(* Logix 5000 project; controller STAT 1756-L72 rev 20.12; software revision 20.04; part 17 of 34 *)
(* tags used below, declared in another part *)
   B14 : DINT[30];
   B16 : DINT[30];
   B17 : DINT[30];
   B3 : DINT[256];
   B9 : DINT[40];
   I7_000_Bit08 : ALIAS FOR I7[0].8;   // midden alarm ketel tampon
   I8_000_Bit09 : ALIAS FOR I8[0].9;   // midden niveau kuip 1 voorb. polyelectrolute
   I8_000_Bit10 : ALIAS FOR I8[0].10;   // hoog niveau kuip 1 voorb. polyelectrolute
   I8_000_Bit12 : ALIAS FOR I8[0].12;   // midden niveau kuip 2 voorb. polyelectrolute
   I8_000_Bit13 : ALIAS FOR I8[0].13;   // hoog niveau pekel
   N26 : DINT[256];
   O12_001_Bit06 : ALIAS FOR O12[1].6;   // TFB1_1_EV1 TFB1_1_EV1
   O12_001_Bit07 : ALIAS FOR O12[1].7;   // TFB1_1_EV2 TFB1_1_EV2
   O12_001_Bit08 : ALIAS FOR O12[1].8;   // TFB1_2_EV3 TFB1_2_EV3
   O12_001_Bit09 : ALIAS FOR O12[1].9;   // TFB1_2_EV4 TFB1_2_EV4
   O12_001_Bit10 : ALIAS FOR O12[1].10;   // TFB1_2_EV10 TFB1_2_EV10
   O12_001_Bit11 : ALIAS FOR O12[1].11;   // TFB1_EV9 TFB1_EV9
   O12_001_Bit12 : ALIAS FOR O12[1].12;   // TFB1_2_EV5 TFB1_2_EV5
   O12_001_Bit13 : ALIAS FOR O12[1].13;   // TFB1_2_EV6 TFB1_2_EV6
   O13_001_Bit10 : ALIAS FOR O13[1].10;   // TFB1_2_EV7 TFB1_2_EV7
   O13_001_Bit11 : ALIAS FOR O13[1].11;   // TFB1_2_EV8 TFB1_2_EV8
   O13_001_Bit12 : ALIAS FOR O13[1].12;   // TFB1_2_EV11 TFB1_2_EV11
   O15_000_Bit09 : ALIAS FOR O15[0].9;   // CLEAN_V11 CLEAN_V11
   O15_000_Bit10 : ALIAS FOR O15[0].10;   // CLEAN_V12 CLEAN_V12
   O15_000_Bit11 : ALIAS FOR O15[0].11;   // CLEAN_V13 CLEAN_V13
   O15_000_Bit12 : ALIAS FOR O15[0].12;   // CLEAN_V14 CLEAN_V14
   O15_000_Bit13 : ALIAS FOR O15[0].13;   // CLEAN_V21 CLEAN_V21
   O15_000_Bit14 : ALIAS FOR O15[0].14;   // CLEAN_V22 CLEAN_V22
   O15_000_Bit15 : ALIAS FOR O15[0].15;   // CLEAN_V23 CLEAN_V23
   O15_001_Bit00 : ALIAS FOR O15[1].0;   // CLEAN_V24 CLEAN_V24
   O15_001_Bit01 : ALIAS FOR O15[1].1;   // CLEAN_V3 CLEAN_V3
   O1_011_Bit00 : ALIAS FOR O1[11].0;
   O1_011_Bit03 : ALIAS FOR O1[11].3;
   STEP_REI_Z_2_3_6_7 : BOOL;
   STEP_REI_Z_2_3_6_7B : BOOL;
   STEP_REO_Z_2_6_A_ET_B : BOOL;
   T4 : TIMER[200];
(* ibt, continued *)

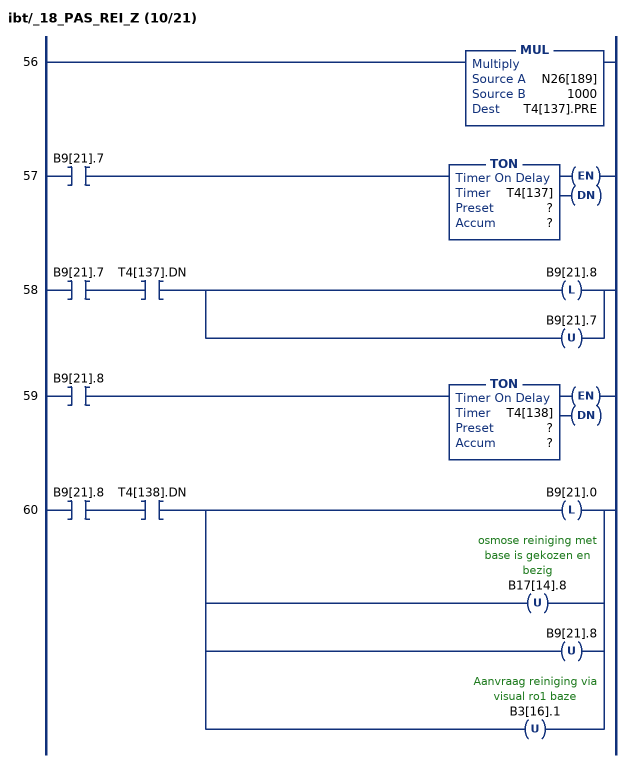
   [picture p297: ibt/_18_PAS_REI_Z rungs 56-60]
   56: MUL(N26[189],1000,T4[137].PRE);
   57: XIC(B9[21].7)TON(T4[137],?,?);
   58: XIC(B9[21].7)XIC(T4[137].DN)[OTL(B9[21].8) ,OTU(B9[21].7) ];
   59: XIC(B9[21].8)TON(T4[138],?,?);
   60: XIC(B9[21].8)XIC(T4[138].DN)[[OTL(B9[21].0) ,OTU(B17[14].8) ] ,[OTU(B9[21].8) ,OTU(B3[16].1) ] ];
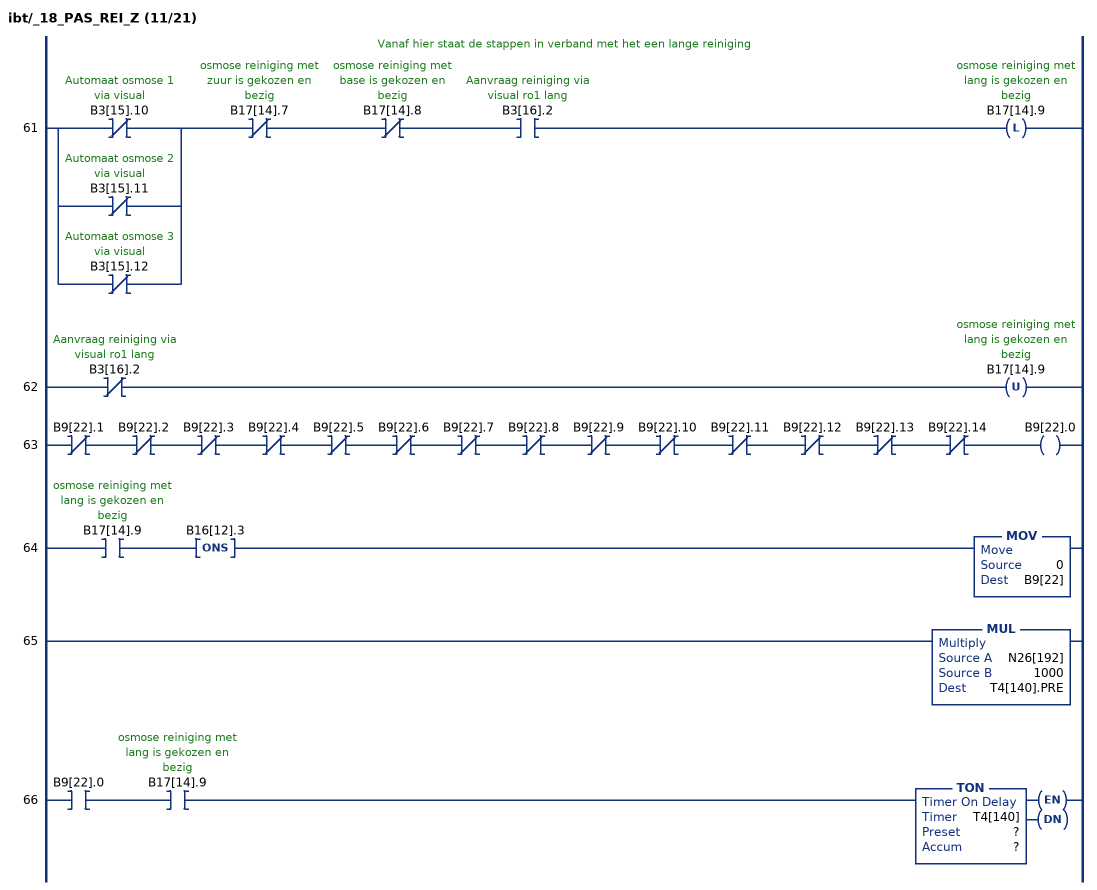
   // Vanaf hier staat de stappen in verband met het een lange reiniging
   61: [XIO(B3[15].10) ,[XIO(B3[15].11) ,XIO(B3[15].12) ] ]XIO(B17[14].7)XIO(B17[14].8)XIC(B3[16].2)OTL(B17[14].9);
   62: XIO(B3[16].2)OTU(B17[14].9);
   63: XIO(B9[22].1)XIO(B9[22].2)XIO(B9[22].3)XIO(B9[22].4)XIO(B9[22].5)XIO(B9[22].6)XIO(B9[22].7)XIO(B9[22].8)XIO(B9[22].9)XIO(B9[22].10)XIO(B9[22].11)XIO(B9[22].12)XIO(B9[22].13)XIO(B9[22].14)OTE(B9[22].0);
   64: XIC(B17[14].9)ONS(B16[12].3)MOV(0,B9[22]);
   65: MUL(N26[192],1000,T4[140].PRE);
   66: XIC(B9[22].0)XIC(B17[14].9)TON(T4[140],?,?);
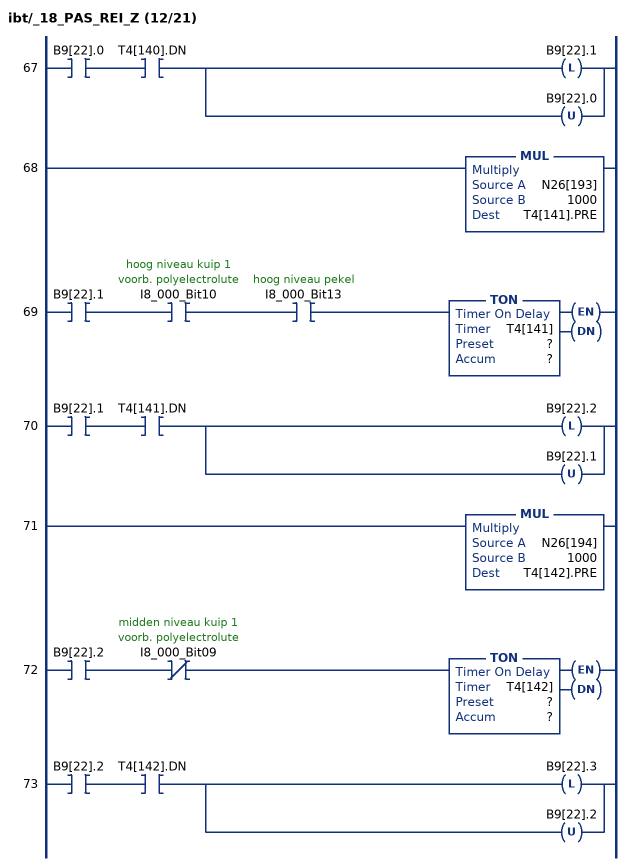
   67: XIC(B9[22].0)XIC(T4[140].DN)[OTL(B9[22].1) ,OTU(B9[22].0) ];
   68: MUL(N26[193],1000,T4[141].PRE);
   69: XIC(B9[22].1)XIC(I8_000_Bit10)XIC(I8_000_Bit13)TON(T4[141],?,?);
   70: XIC(B9[22].1)XIC(T4[141].DN)[OTL(B9[22].2) ,OTU(B9[22].1) ];
   71: MUL(N26[194],1000,T4[142].PRE);
   72: XIC(B9[22].2)XIO(I8_000_Bit09)TON(T4[142],?,?);
   73: XIC(B9[22].2)XIC(T4[142].DN)[OTL(B9[22].3) ,OTU(B9[22].2) ];
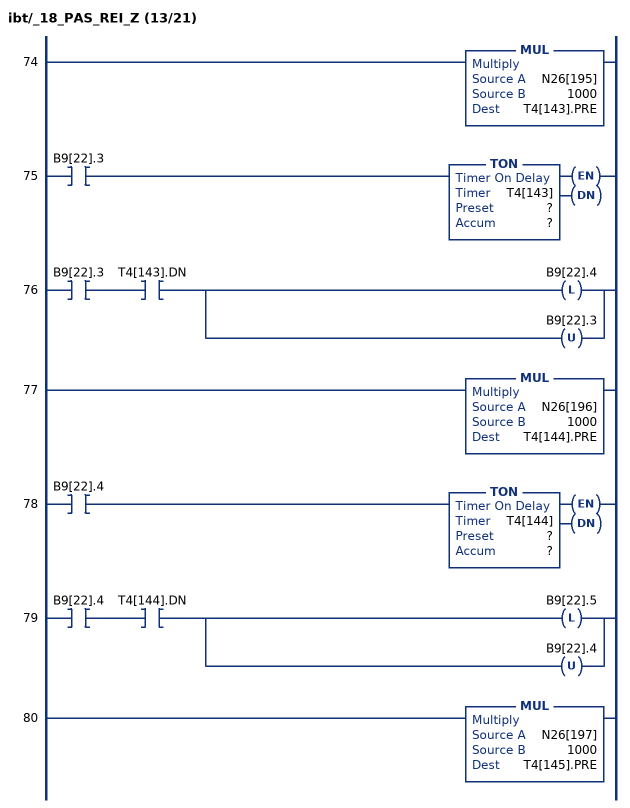
   74: MUL(N26[195],1000,T4[143].PRE);
   75: XIC(B9[22].3)TON(T4[143],?,?);
   76: XIC(B9[22].3)XIC(T4[143].DN)[OTL(B9[22].4) ,OTU(B9[22].3) ];
   77: MUL(N26[196],1000,T4[144].PRE);
   78: XIC(B9[22].4)TON(T4[144],?,?);
   79: XIC(B9[22].4)XIC(T4[144].DN)[OTL(B9[22].5) ,OTU(B9[22].4) ];
   80: MUL(N26[197],1000,T4[145].PRE);
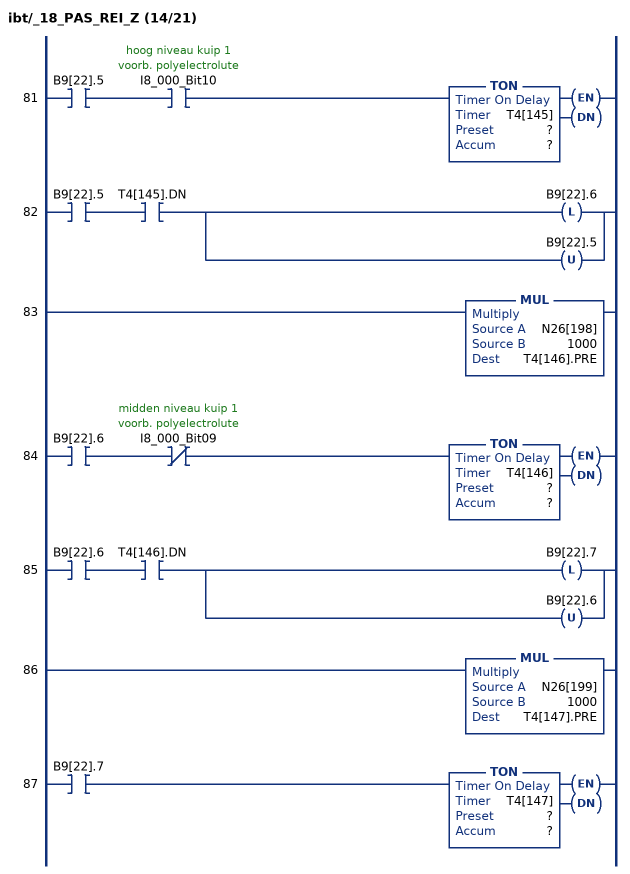
   81: XIC(B9[22].5)XIC(I8_000_Bit10)TON(T4[145],?,?);
   82: XIC(B9[22].5)XIC(T4[145].DN)[OTL(B9[22].6) ,OTU(B9[22].5) ];
   83: MUL(N26[198],1000,T4[146].PRE);
   84: XIC(B9[22].6)XIO(I8_000_Bit09)TON(T4[146],?,?);
   85: XIC(B9[22].6)XIC(T4[146].DN)[OTL(B9[22].7) ,OTU(B9[22].6) ];
   86: MUL(N26[199],1000,T4[147].PRE);
   87: XIC(B9[22].7)TON(T4[147],?,?);
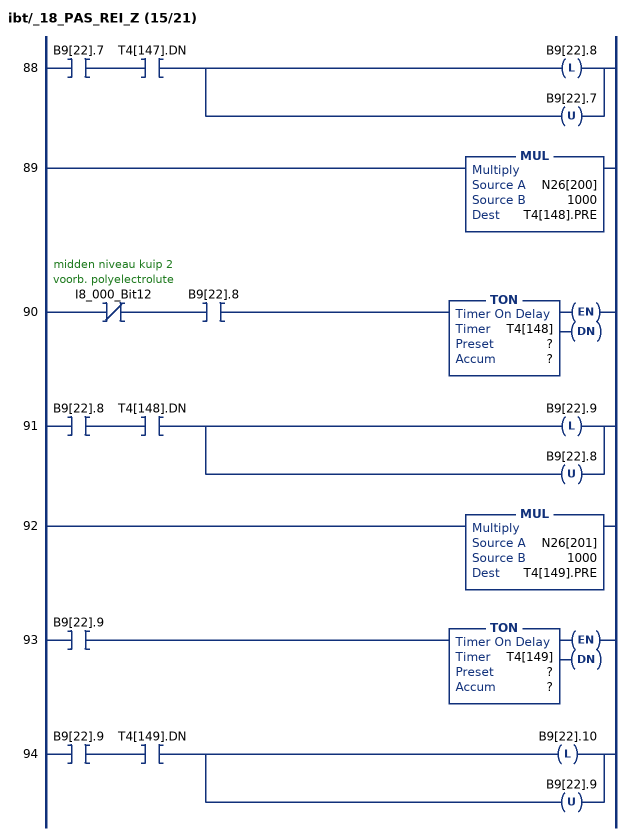
   88: XIC(B9[22].7)XIC(T4[147].DN)[OTL(B9[22].8) ,OTU(B9[22].7) ];
   89: MUL(N26[200],1000,T4[148].PRE);
   90: XIO(I8_000_Bit12)XIC(B9[22].8)TON(T4[148],?,?);
   91: XIC(B9[22].8)XIC(T4[148].DN)[OTL(B9[22].9) ,OTU(B9[22].8) ];
   92: MUL(N26[201],1000,T4[149].PRE);
   93: XIC(B9[22].9)TON(T4[149],?,?);
   94: XIC(B9[22].9)XIC(T4[149].DN)[OTL(B9[22].10) ,OTU(B9[22].9) ];
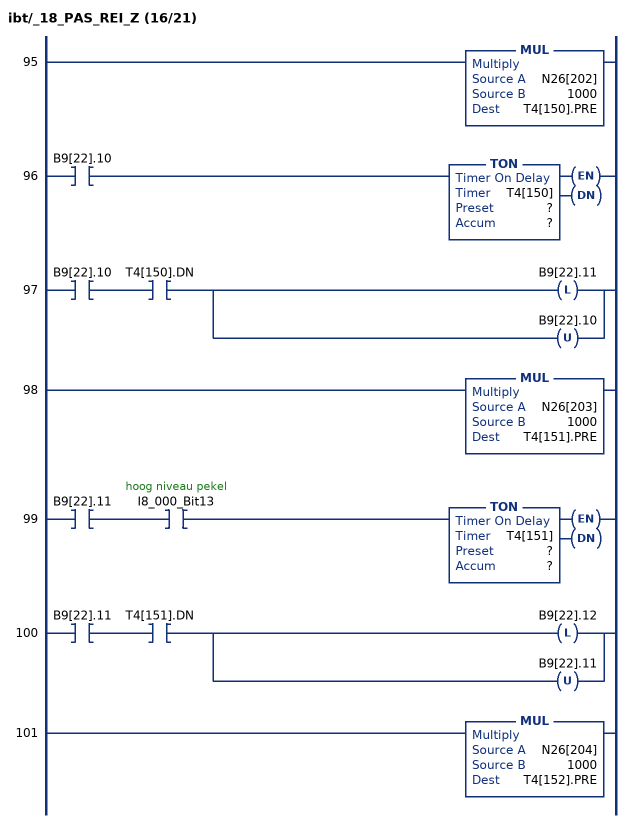
   95: MUL(N26[202],1000,T4[150].PRE);
   96: XIC(B9[22].10)TON(T4[150],?,?);
   97: XIC(B9[22].10)XIC(T4[150].DN)[OTL(B9[22].11) ,OTU(B9[22].10) ];
   98: MUL(N26[203],1000,T4[151].PRE);
   99: XIC(B9[22].11)XIC(I8_000_Bit13)TON(T4[151],?,?);
   100: XIC(B9[22].11)XIC(T4[151].DN)[OTL(B9[22].12) ,OTU(B9[22].11) ];
   101: MUL(N26[204],1000,T4[152].PRE);
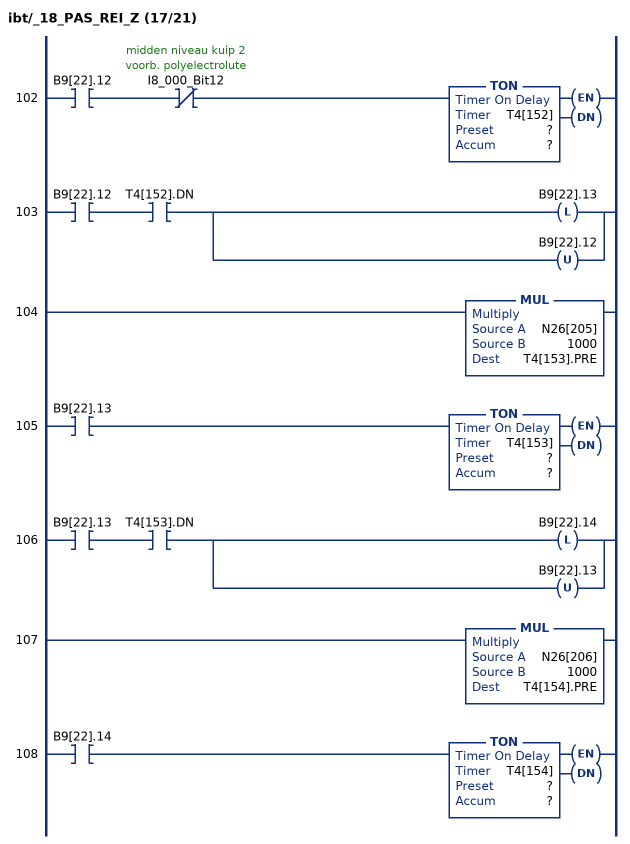
   102: XIC(B9[22].12)XIO(I8_000_Bit12)TON(T4[152],?,?);
   103: XIC(B9[22].12)XIC(T4[152].DN)[OTL(B9[22].13) ,OTU(B9[22].12) ];
   104: MUL(N26[205],1000,T4[153].PRE);
   105: XIC(B9[22].13)TON(T4[153],?,?);
   106: XIC(B9[22].13)XIC(T4[153].DN)[OTL(B9[22].14) ,OTU(B9[22].13) ];
   107: MUL(N26[206],1000,T4[154].PRE);
   108: XIC(B9[22].14)TON(T4[154],?,?);
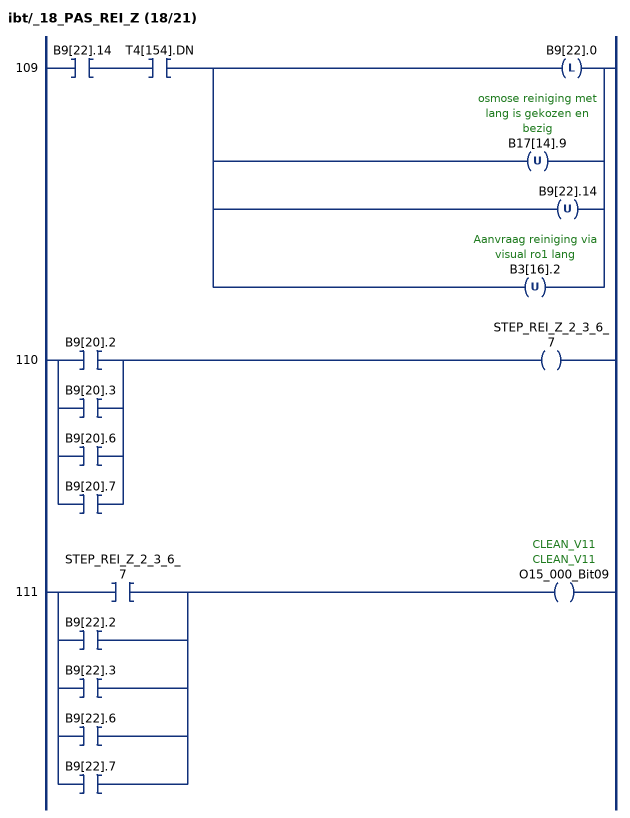
   109: XIC(B9[22].14)XIC(T4[154].DN)[[OTL(B9[22].0) ,OTU(B17[14].9) ] ,[OTU(B9[22].14) ,OTU(B3[16].2) ] ];
   110: [XIC(B9[20].2) ,[XIC(B9[20].3) ,[XIC(B9[20].6) ,XIC(B9[20].7) ] ] ]OTE(STEP_REI_Z_2_3_6_7);
   111: [XIC(STEP_REI_Z_2_3_6_7) ,[[XIC(B9[22].2) ,XIC(B9[22].3) ] ,[XIC(B9[22].6) ,XIC(B9[22].7) ] ] ]OTE(O15_000_Bit09);
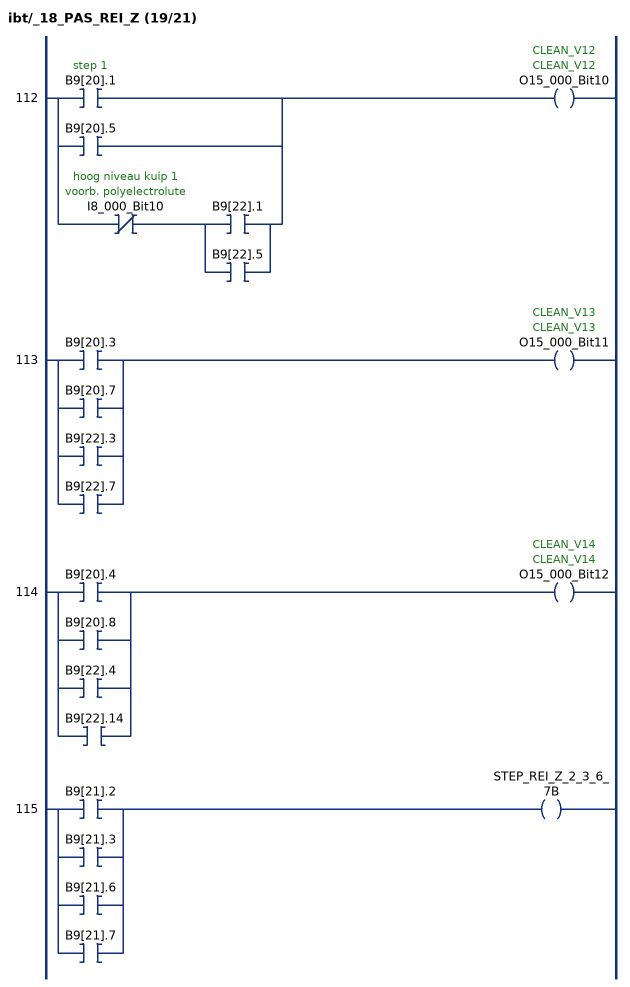
   112: [[XIC(B9[20].1) ,XIC(B9[20].5) ] ,XIO(I8_000_Bit10) [XIC(B9[22].1) ,XIC(B9[22].5) ] ]OTE(O15_000_Bit10);
   113: [[XIC(B9[20].3) ,XIC(B9[20].7) ] ,[XIC(B9[22].3) ,XIC(B9[22].7) ] ]OTE(O15_000_Bit11);
   114: [[XIC(B9[20].4) ,XIC(B9[20].8) ] ,[XIC(B9[22].4) ,XIC(B9[22].14) ] ]OTE(O15_000_Bit12);
   115: [[XIC(B9[21].2) ,XIC(B9[21].3) ] ,[XIC(B9[21].6) ,XIC(B9[21].7) ] ]OTE(STEP_REI_Z_2_3_6_7B);
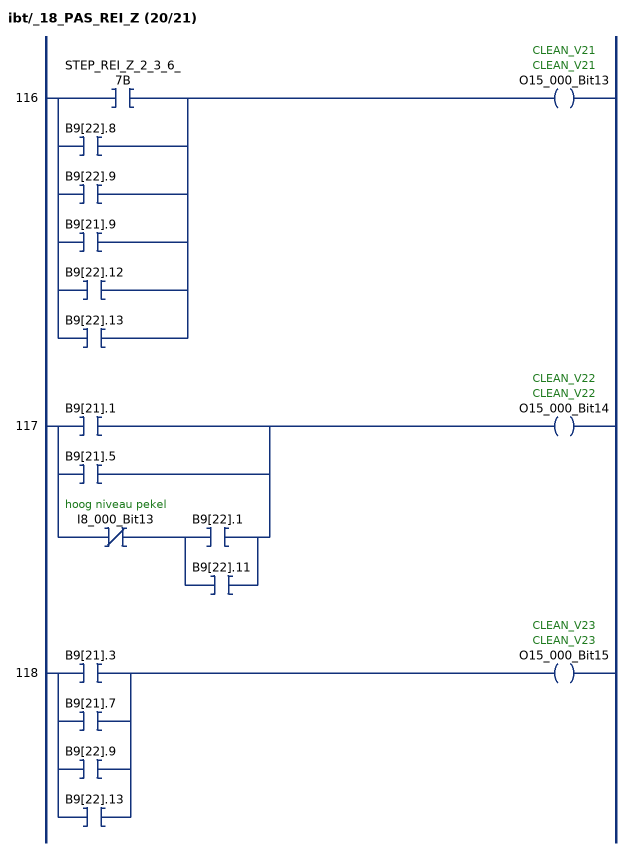
   116: [[XIC(STEP_REI_Z_2_3_6_7B) ,XIC(B9[22].8) ,XIC(B9[22].9) ] ,[XIC(B9[21].9) ,[XIC(B9[22].12) ,XIC(B9[22].13) ] ] ]OTE(O15_000_Bit13);
   117: [[XIC(B9[21].1) ,XIC(B9[21].5) ] ,XIO(I8_000_Bit13) [XIC(B9[22].1) ,XIC(B9[22].11) ] ]OTE(O15_000_Bit14);
   118: [[XIC(B9[21].3) ,XIC(B9[21].7) ] ,[XIC(B9[22].9) ,XIC(B9[22].13) ] ]OTE(O15_000_Bit15);
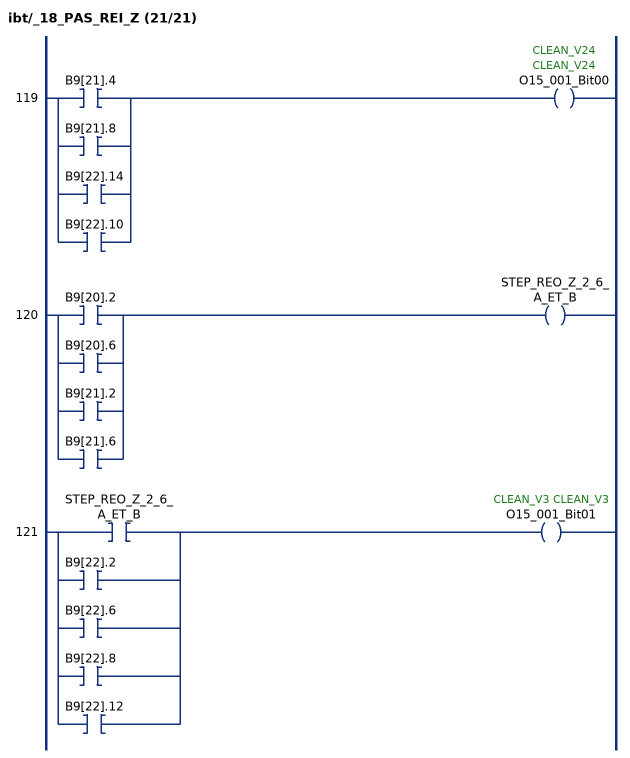
   119: [[XIC(B9[21].4) ,XIC(B9[21].8) ] ,XIC(B9[22].14) ,XIC(B9[22].10) ]OTE(O15_001_Bit00);
   120: [[XIC(B9[20].2) ,[XIC(B9[20].6) ,XIC(B9[21].2) ] ] ,XIC(B9[21].6) ]OTE(STEP_REO_Z_2_6_A_ET_B);
   121: [[XIC(STEP_REO_Z_2_6_A_ET_B) ,[XIC(B9[22].2) ,XIC(B9[22].6) ] ] ,[XIC(B9[22].8) ,XIC(B9[22].12) ] ]OTE(O15_001_Bit01);
END_ROUTINE

ROUTINE _19_SEQ_ONTEIZ   (* ladder *)
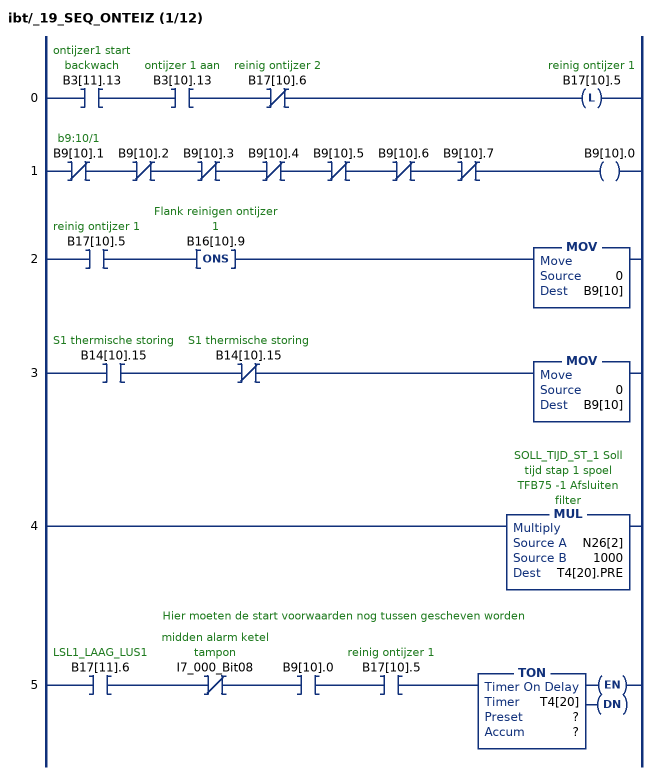
   0: XIC(B3[11].13)XIC(B3[10].13)XIO(B17[10].6)OTL(B17[10].5);
   1: XIO(B9[10].1)XIO(B9[10].2)XIO(B9[10].3)XIO(B9[10].4)XIO(B9[10].5)XIO(B9[10].6)XIO(B9[10].7)OTE(B9[10].0);
   2: XIC(B17[10].5)ONS(B16[10].9)MOV(0,B9[10]);
   3: XIC(B14[10].15)XIO(B14[10].15)MOV(0,B9[10]);
   4: MUL(N26[2],1000,T4[20].PRE);
   // Hier moeten de start voorwaarden nog tussen gescheven worden
   5: XIC(B17[11].6)XIO(I7_000_Bit08)XIC(B9[10].0)XIC(B17[10].5)TON(T4[20],?,?);
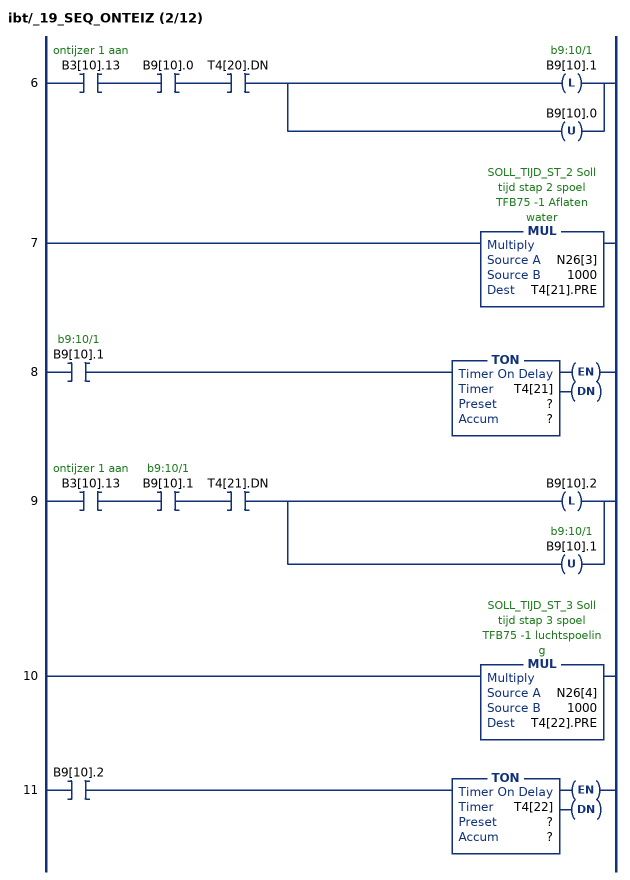
   6: XIC(B3[10].13)XIC(B9[10].0)XIC(T4[20].DN)[OTL(B9[10].1) ,OTU(B9[10].0) ];
   7: MUL(N26[3],1000,T4[21].PRE);
   8: XIC(B9[10].1)TON(T4[21],?,?);
   9: XIC(B3[10].13)XIC(B9[10].1)XIC(T4[21].DN)[OTL(B9[10].2) ,OTU(B9[10].1) ];
   10: MUL(N26[4],1000,T4[22].PRE);
   11: XIC(B9[10].2)TON(T4[22],?,?);
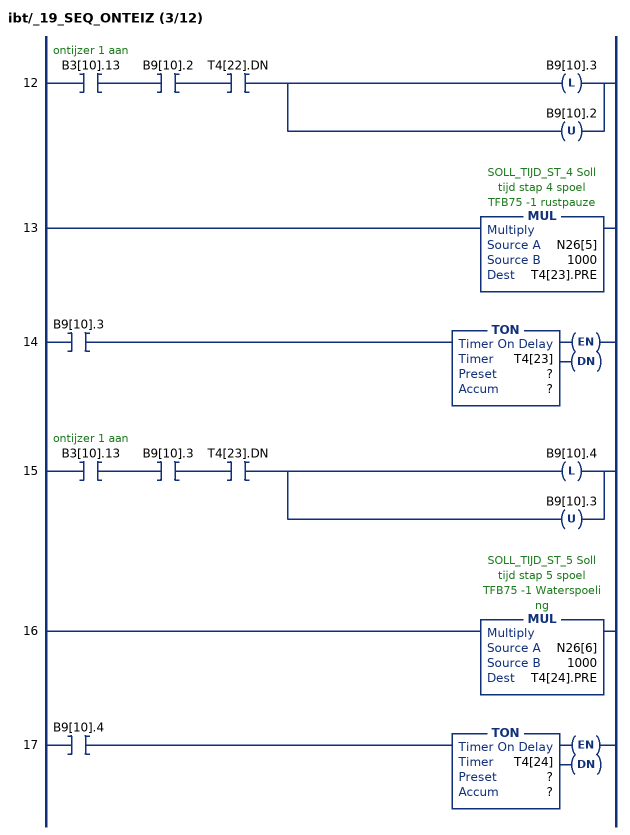
   12: XIC(B3[10].13)XIC(B9[10].2)XIC(T4[22].DN)[OTL(B9[10].3) ,OTU(B9[10].2) ];
   13: MUL(N26[5],1000,T4[23].PRE);
   14: XIC(B9[10].3)TON(T4[23],?,?);
   15: XIC(B3[10].13)XIC(B9[10].3)XIC(T4[23].DN)[OTL(B9[10].4) ,OTU(B9[10].3) ];
   16: MUL(N26[6],1000,T4[24].PRE);
   17: XIC(B9[10].4)TON(T4[24],?,?);
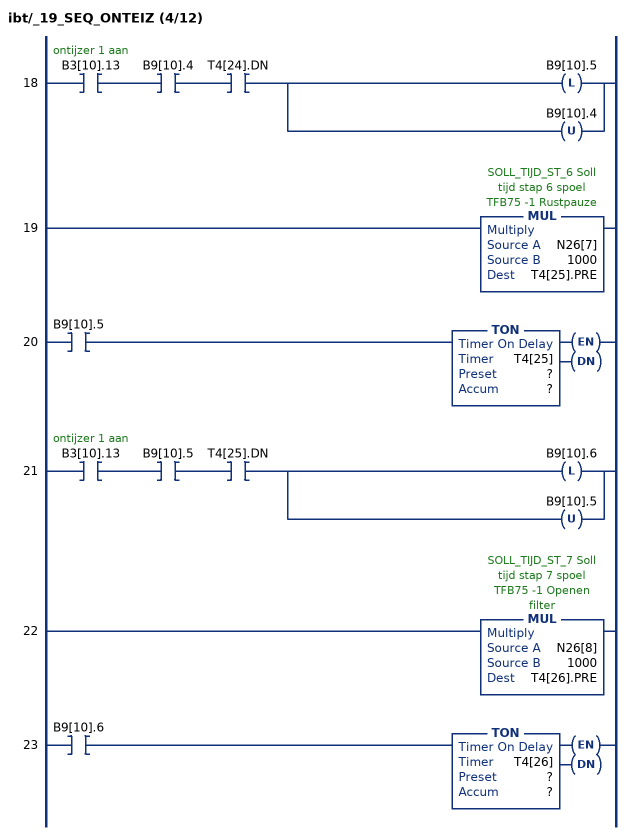
   18: XIC(B3[10].13)XIC(B9[10].4)XIC(T4[24].DN)[OTL(B9[10].5) ,OTU(B9[10].4) ];
   19: MUL(N26[7],1000,T4[25].PRE);
   20: XIC(B9[10].5)TON(T4[25],?,?);
   21: XIC(B3[10].13)XIC(B9[10].5)XIC(T4[25].DN)[OTL(B9[10].6) ,OTU(B9[10].5) ];
   22: MUL(N26[8],1000,T4[26].PRE);
   23: XIC(B9[10].6)TON(T4[26],?,?);
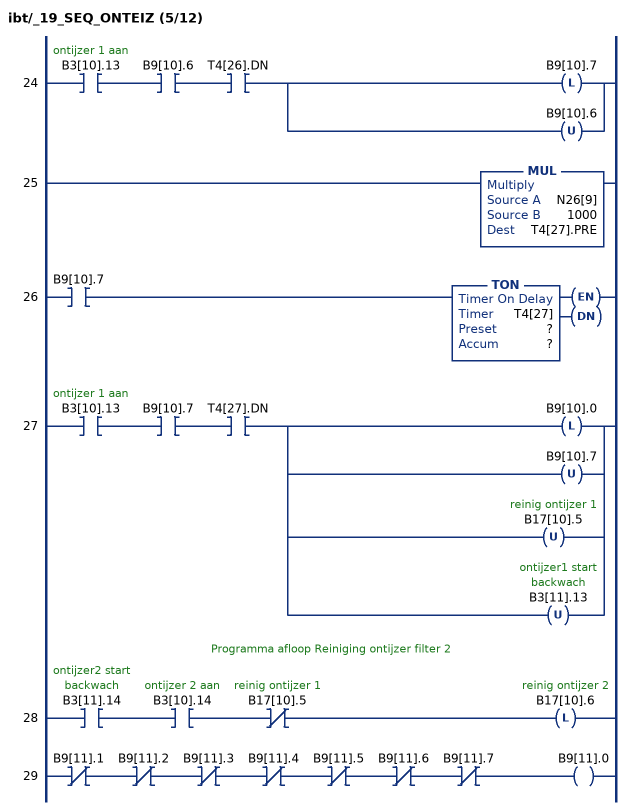
   24: XIC(B3[10].13)XIC(B9[10].6)XIC(T4[26].DN)[OTL(B9[10].7) ,OTU(B9[10].6) ];
   25: MUL(N26[9],1000,T4[27].PRE);
   26: XIC(B9[10].7)TON(T4[27],?,?);
   27: XIC(B3[10].13)XIC(B9[10].7)XIC(T4[27].DN)[OTL(B9[10].0) ,[OTU(B9[10].7) ,[OTU(B17[10].5) ,OTU(B3[11].13) ] ] ];
   // Programma afloop Reiniging ontijzer filter 2
   28: XIC(B3[11].14)XIC(B3[10].14)XIO(B17[10].5)OTL(B17[10].6);
   29: XIO(B9[11].1)XIO(B9[11].2)XIO(B9[11].3)XIO(B9[11].4)XIO(B9[11].5)XIO(B9[11].6)XIO(B9[11].7)OTE(B9[11].0);
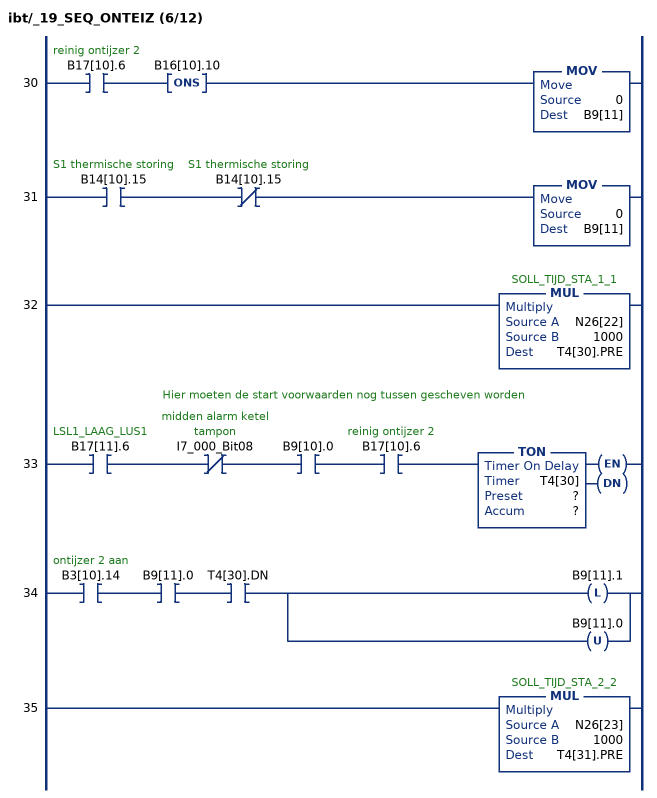
   30: XIC(B17[10].6)ONS(B16[10].10)MOV(0,B9[11]);
   31: XIC(B14[10].15)XIO(B14[10].15)MOV(0,B9[11]);
   32: MUL(N26[22],1000,T4[30].PRE);
   // Hier moeten de start voorwaarden nog tussen gescheven worden
   33: XIC(B17[11].6)XIO(I7_000_Bit08)XIC(B9[10].0)XIC(B17[10].6)TON(T4[30],?,?);
   34: XIC(B3[10].14)XIC(B9[11].0)XIC(T4[30].DN)[OTL(B9[11].1) ,OTU(B9[11].0) ];
   35: MUL(N26[23],1000,T4[31].PRE);
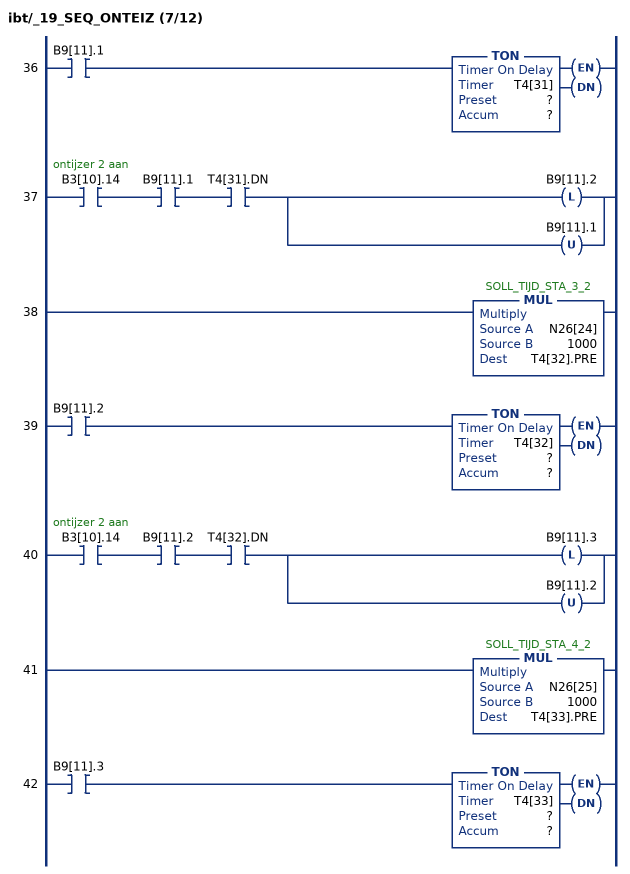
   36: XIC(B9[11].1)TON(T4[31],?,?);
   37: XIC(B3[10].14)XIC(B9[11].1)XIC(T4[31].DN)[OTL(B9[11].2) ,OTU(B9[11].1) ];
   38: MUL(N26[24],1000,T4[32].PRE);
   39: XIC(B9[11].2)TON(T4[32],?,?);
   40: XIC(B3[10].14)XIC(B9[11].2)XIC(T4[32].DN)[OTL(B9[11].3) ,OTU(B9[11].2) ];
   41: MUL(N26[25],1000,T4[33].PRE);
   42: XIC(B9[11].3)TON(T4[33],?,?);
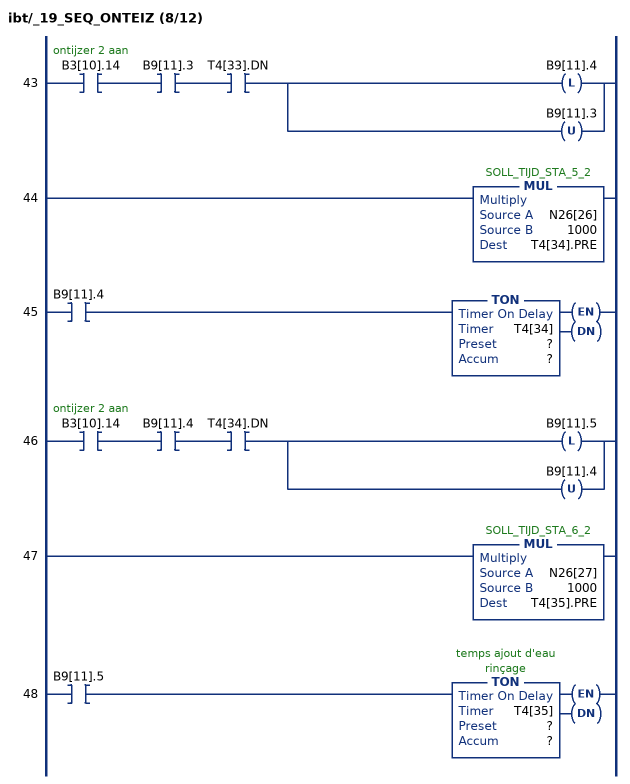
   43: XIC(B3[10].14)XIC(B9[11].3)XIC(T4[33].DN)[OTL(B9[11].4) ,OTU(B9[11].3) ];
   44: MUL(N26[26],1000,T4[34].PRE);
   45: XIC(B9[11].4)TON(T4[34],?,?);
   46: XIC(B3[10].14)XIC(B9[11].4)XIC(T4[34].DN)[OTL(B9[11].5) ,OTU(B9[11].4) ];
   47: MUL(N26[27],1000,T4[35].PRE);
   48: XIC(B9[11].5)TON(T4[35],?,?);
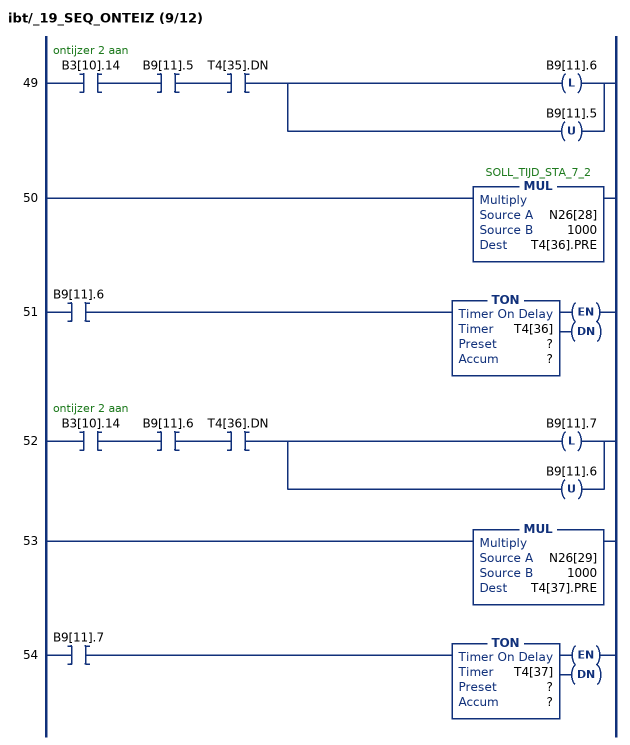
   49: XIC(B3[10].14)XIC(B9[11].5)XIC(T4[35].DN)[OTL(B9[11].6) ,OTU(B9[11].5) ];
   50: MUL(N26[28],1000,T4[36].PRE);
   51: XIC(B9[11].6)TON(T4[36],?,?);
   52: XIC(B3[10].14)XIC(B9[11].6)XIC(T4[36].DN)[OTL(B9[11].7) ,OTU(B9[11].6) ];
   53: MUL(N26[29],1000,T4[37].PRE);
   54: XIC(B9[11].7)TON(T4[37],?,?);
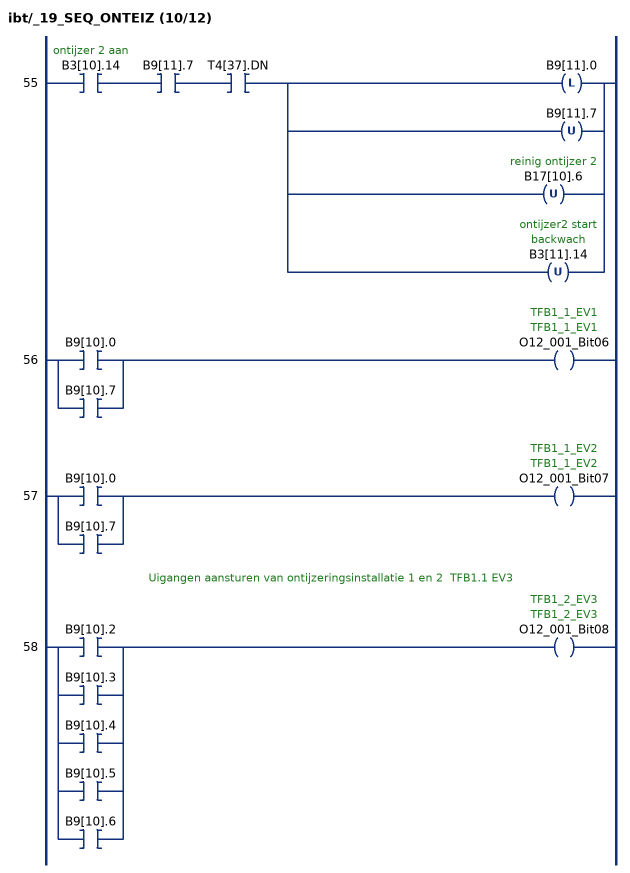
   55: XIC(B3[10].14)XIC(B9[11].7)XIC(T4[37].DN)[OTL(B9[11].0) ,[OTU(B9[11].7) ,[OTU(B17[10].6) ,OTU(B3[11].14) ] ] ];
   56: [XIC(B9[10].0) ,XIC(B9[10].7) ]OTE(O12_001_Bit06);
   57: [XIC(B9[10].0) ,XIC(B9[10].7) ]OTE(O12_001_Bit07);
   // Uigangen aansturen van ontijzeringsinstallatie 1 en 2  TFB1.1 EV3
   58: [XIC(B9[10].2) ,[XIC(B9[10].3) ,[XIC(B9[10].4) ,[XIC(B9[10].5) ,XIC(B9[10].6) ] ] ] ]OTE(O12_001_Bit08);
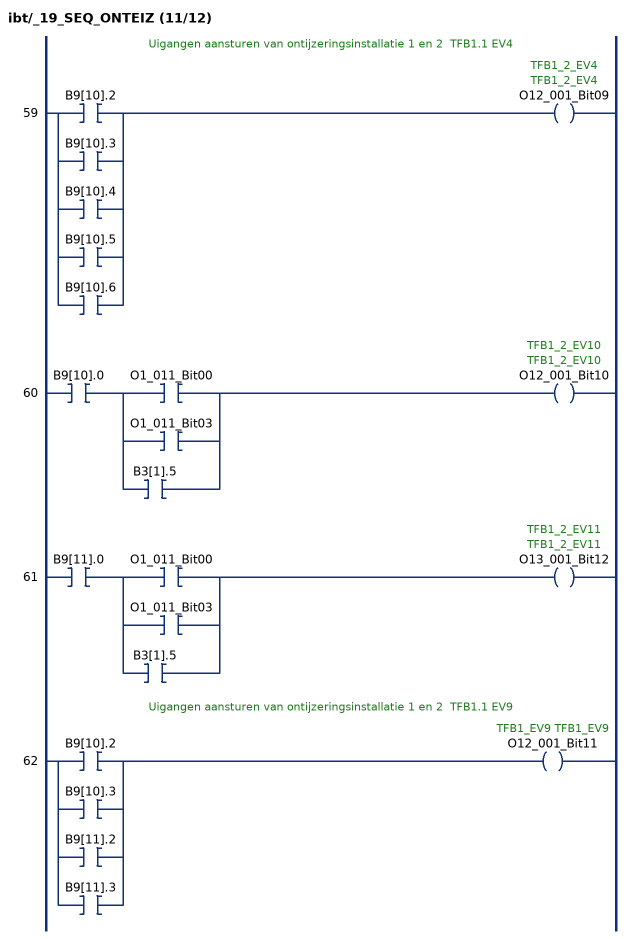
   // Uigangen aansturen van ontijzeringsinstallatie 1 en 2  TFB1.1 EV4
   59: [XIC(B9[10].2) ,[XIC(B9[10].3) ,[XIC(B9[10].4) ,[XIC(B9[10].5) ,XIC(B9[10].6) ] ] ] ]OTE(O12_001_Bit09);
   60: XIC(B9[10].0)[XIC(O1_011_Bit00) ,XIC(O1_011_Bit03) ,XIC(B3[1].5) ]OTE(O12_001_Bit10);
   61: XIC(B9[11].0)[XIC(O1_011_Bit00) ,XIC(O1_011_Bit03) ,XIC(B3[1].5) ]OTE(O13_001_Bit12);
   // Uigangen aansturen van ontijzeringsinstallatie 1 en 2  TFB1.1 EV9
   62: [XIC(B9[10].2) ,[XIC(B9[10].3) ,[XIC(B9[11].2) ,XIC(B9[11].3) ] ] ]OTE(O12_001_Bit11);
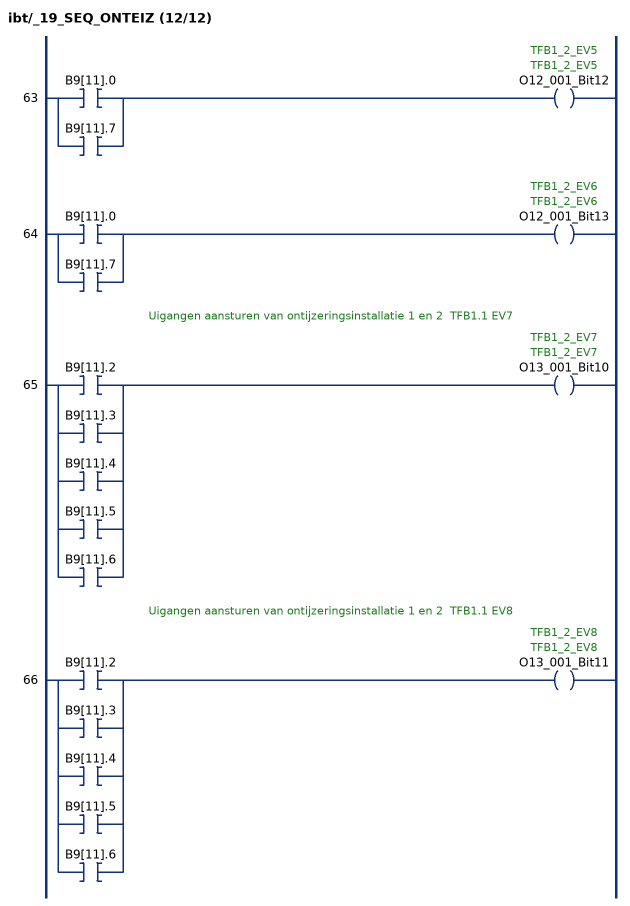
   63: [XIC(B9[11].0) ,XIC(B9[11].7) ]OTE(O12_001_Bit12);
   64: [XIC(B9[11].0) ,XIC(B9[11].7) ]OTE(O12_001_Bit13);
   // Uigangen aansturen van ontijzeringsinstallatie 1 en 2  TFB1.1 EV7
   65: [XIC(B9[11].2) ,[XIC(B9[11].3) ,[XIC(B9[11].4) ,[XIC(B9[11].5) ,XIC(B9[11].6) ] ] ] ]OTE(O13_001_Bit10);
   // Uigangen aansturen van ontijzeringsinstallatie 1 en 2  TFB1.1 EV8
   66: [XIC(B9[11].2) ,[XIC(B9[11].3) ,[XIC(B9[11].4) ,[XIC(B9[11].5) ,XIC(B9[11].6) ] ] ] ]OTE(O13_001_Bit11);
END_ROUTINE
